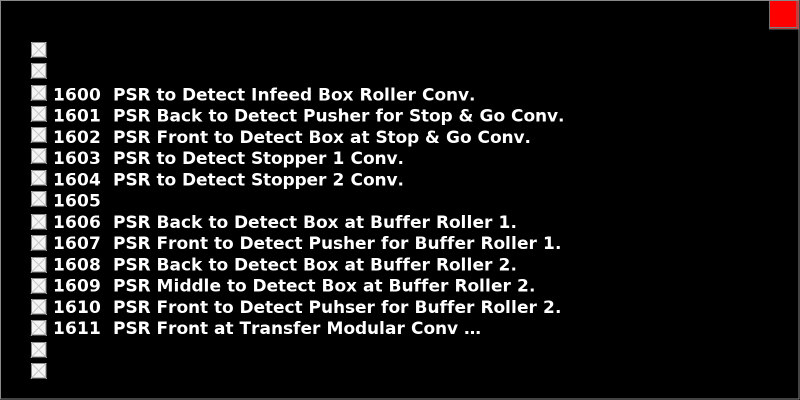
VISUALIZATION P2_DI7  // 800x400, background image 
    ImageSwitcher (31,42 15x15), variable: InputOutput_GVL.Digital_Input[97], behaviour: TOGGLE
    Label (50,16 696x391), "1600 PSR to Detect Infeed Box Roller Conv. 1601 PSR Back to Detect Pusher for Stop & Go Conv. 1602 PSR Front to Detect Box at Stop & Go Conv. 1603 PSR to Detect Stopper 1 Conv. 1604 PSR to Detect Stopper 2 Conv. 1605 1606 PSR Back to Detect Box at Buffer Roller 1. 1607 PSR Front to Detect Pusher for Buffer Roller 1. 1608 PSR Back to Detect Box at Buffer Roller 2. 1609 PSR Middle to Detect Box at Buffer Roller 2. 1610 PSR Front to Detect Puhser for Buffer Roller 2. 1611 PSR Front at Transfer Modular Conv 4 1612 PSR Front at Transfer Modular Conv 2 1613 PSR Back at Transfer Modular Conv 3 1614 PSR Front at Transfer Modular Conv 3 1615 PSR Back at Transfer Modular Conv 4"
    ImageSwitcher (31,63 15x15), variable: InputOutput_GVL.Digital_Input[98], behaviour: TOGGLE
    ImageSwitcher (31,85 15x15), variable: InputOutput_GVL.Digital_Input[99], behaviour: TOGGLE
    ImageSwitcher (31,106 15x15), variable: InputOutput_GVL.Digital_Input[100], behaviour: TOGGLE
    ImageSwitcher (31,127 15x15), variable: InputOutput_GVL.Digital_Input[101], behaviour: TOGGLE
    ImageSwitcher (31,148 15x15), variable: InputOutput_GVL.Digital_Input[102], behaviour: TOGGLE
    ImageSwitcher (31,170 15x15), variable: InputOutput_GVL.Digital_Input[103], behaviour: TOGGLE
    ImageSwitcher (31,191 15x15), variable: InputOutput_GVL.Digital_Input[104], behaviour: TOGGLE
    ImageSwitcher (31,214 15x15), variable: InputOutput_GVL.Digital_Input[105], behaviour: TOGGLE
    ImageSwitcher (31,235 15x15), variable: InputOutput_GVL.Digital_Input[106], behaviour: TOGGLE
    ImageSwitcher (31,257 15x15), variable: InputOutput_GVL.Digital_Input[107], behaviour: TOGGLE
    ImageSwitcher (31,278 15x15), variable: InputOutput_GVL.Digital_Input[108], behaviour: TOGGLE
    ImageSwitcher (31,299 15x15), variable: InputOutput_GVL.Digital_Input[109], behaviour: TOGGLE
    ImageSwitcher (31,320 15x15), variable: InputOutput_GVL.Digital_Input[110], behaviour: TOGGLE
    ImageSwitcher (31,342 15x15), variable: InputOutput_GVL.Digital_Input[111], behaviour: TOGGLE
    ImageSwitcher (31,363 15x15), variable: InputOutput_GVL.Digital_Input[112], behaviour: TOGGLE
    Button (769,-1 30x30), image: VisuSymbols.Symbols.Wrong
        OnMouseClick: CloseDialog Dialog=P2_DI7, Result=OK, NumpadKeypadSet=True
END_VISUALIZATION

(* stored: Version 1.1.0.1, ProductVersion 3.1.4024.12
   Visu P2_DI7: Id {8bc09e45-a270-45da-bedd-e79b92cf50df} *)
